// TIA Portal V20 export
// export: Created 2025-12-01T14:57:47.0697469Z, ExportSetting None, DisplayName Totally Integrated Automation Portal, DisplayVersion V20 Update 3, DisplayName TIA Portal Openness, DisplayVersion V20 Update 3, DisplayName TIA Portal Version Control Interface, DisplayVersion V20 Update 3, DisplayName STEP 7 Professional, DisplayVersion V20 Update 3, DisplayName STEP 7 Safety, DisplayVersion V20 Update 2, DisplayName WinCC Basic/Comfort/Advanced, DisplayVersion V20 Update 3, DisplayName WinCC Professional, DisplayVersion V20 Update 3, DisplayName WinCC Unified, DisplayVersion V20 Update 3
FUNCTION "FC522_Buc_Busc_Etiquetas" : Void   // FC522, LAD
{ S7_Optimized_Access := 'FALSE' }
AUTHOR : ROUTER
NAME : 20130623
VERSION : 3.1
// stored: AutoNumber false, SetENOAutomatically false
   VAR_TEMP
      Valor_Etiqueta : ULInt;
      CNT_Scanner : UInt;
      CNT_Caracter_Etiqueta : UInt;
      Peso_caracter : ULInt;
      bucle_scanners : Bool;
      Fin_conversion : Bool;
      contador : UInt;
   END_VAR
BEGIN

REGION Network 1 (SCL)
   REGION inicializacion
       #Valor_Etiqueta := 0;
       #Peso_caracter := 1;
       #CNT_Caracter_Etiqueta := "ROUT_Long_Etiqueta" - 1;
       #CNT_Scanner := 1;
       #bucle_scanners := 1;
   END_REGION
END_REGION

REGION Network 2 (SCL)
   WHILE #bucle_scanners DO
       IF "DB211_Lecturas_Scanner".Lec_Scanner[#CNT_Scanner].Lectura_SCR[0] = 'N' THEN
           // convertir lectura iniciamos el bucle de conversión
           #contador := #CNT_Caracter_Etiqueta;
           #Valor_Etiqueta := 0;
           #Peso_caracter := 1;
           #Fin_conversion := 0;
           WHILE (NOT (#Fin_conversion)) DO
               IF (("DB211_Lecturas_Scanner".Lec_Scanner[#CNT_Scanner].Lectura_SCR[#contador] >= '0') AND ("DB211_Lecturas_Scanner".Lec_Scanner[#CNT_Scanner].Lectura_SCR[#contador] <= '9')) THEN
                   #Valor_Etiqueta += ((CHAR_TO_INT("DB211_Lecturas_Scanner".Lec_Scanner[#CNT_Scanner].Lectura_SCR[#contador])-48)* #Peso_caracter);
                   #contador -= 1;
                   #Peso_caracter *= 10;
               ELSE
                   #Fin_conversion := true;
                   "DB211_Lecturas_Scanner".Lec_Scanner[#CNT_Scanner].Lectura_SCR[0] := L#0;
                   // ya hemos terminado de convertir el valor, buscamos la etiqueta
              "FC716_Router_BuscarEtiqueta_Lint_y_sacar_orden"(Etiqueta := #Valor_Etiqueta,
                                                                    Numero_SCR := #CNT_Scanner);

               END_IF;

           END_WHILE;


       ELSE // pasar al siguiente scanenr
           #CNT_Scanner += 1;
           IF #CNT_Scanner <= "ROUT_Max_Scanners" THEN
               ;
           ELSE
               RETURN;
           END_IF;
       END_IF;
   END_WHILE;
END_REGION
END_FUNCTION
